PROGRAM MAIN
VAR
END_VAR

IF Estop THEN
	Safety_Ok := FALSE;
END_IF
IF Fault_Reset THEN
	Safety_Ok := TRUE;
END_IF
IF Safety_Ok THEN
Master_On := TRUE;
END_IF
IF Master_On THEN
Auto_Cycle_Fix1();
Auto_Cycle_Fix2();
END_IF

END_PROGRAM

(* stored: Version 1.1.0.1, ProductVersion 3.1.4024.16
   POU MAIN: Id {979b4bbd-69e2-489e-a91d-c2f54e55c89f}, SpecialFunc None *)
